// Mitsubishi GX Works2 project: PLC_GROUP2   PLC: FX3G

// global labels: Global1
VAR_GLOBAL
  SW10 AT X010 : BOOL;
END_VAR
VAR_GLOBAL CONSTANT
  chocolate : REAL := 1200;
  nuts : REAL := 300;
END_VAR
VAR_GLOBAL
  Dnuts AT D3100 : REAL;
END_VAR
VAR_GLOBAL CONSTANT
  pist : REAL := 300;
END_VAR
VAR_GLOBAL
  Dpist AT D3200 : REAL;
END_VAR
VAR_GLOBAL CONSTANT
  kad : REAL := 120;
END_VAR
VAR_GLOBAL
  SW1 AT X001 : BOOL;
  LAMP1 AT Y001 : BOOL;
END_VAR
VAR_GLOBAL CONSTANT
  melt_conts : REAL := 400;
END_VAR
VAR_GLOBAL
  Dchoco AT D3000 : REAL;
  Dkad AT D3300 : REAL;
END_VAR
VAR_GLOBAL CONSTANT
  meltTime : INT := 45;
END_VAR
VAR_GLOBAL
  meltingIndicator AT Y001 : BOOL;
  meltCoil AT TC1 : BOOL;
  SW07 AT X007 : BOOL;
  DAY_STARTED AT Y007 : BOOL;
  Dmelt AT D3400 : REAL;
  meltingprocess AT Y001 : BOOL;
  timeend AT M1 : BOOL;
  Dchocofill AT D2000 : REAL;
  Dnutsfill AT D2010 : REAL;
  Dpistfill AT D2020 : REAL;
  Dkadfill AT D2030 : REAL;
  StartDay AT Y007 : BOOL;
  shutDown AT X005 : BOOL;
  melting AT Y001 : BOOL;
  maxTemp AT X002 : BOOL;
  Lowchoco AT Y007 : BOOL;
  moldsCheck AT X003 : BOOL;
  moldCounter AT CC1 : BOOL;
END_VAR
VAR_GLOBAL CONSTANT
  CValue : INT := 4;
END_VAR
VAR_GLOBAL
  moldsIndicator AT CS1 : BOOL;
  castIndicator AT TS1 : BOOL;
END_VAR
VAR_GLOBAL CONSTANT
  castingTime : INT := 50;
END_VAR
VAR_GLOBAL
  casting AT Y002 : BOOL;
  movedToCasting AT M2 : BOOL;
  finishedCsting AT M3 : BOOL;
END_VAR
VAR_GLOBAL CONSTANT
  CastTime : WORD := 40;
END_VAR
VAR_GLOBAL
  cremeFilling AT X004 : BOOL;
  save_analog_1 AT D8201 : REAL;
END_VAR
VAR_GLOBAL CONSTANT
  input : REAL := 5;
END_VAR
VAR_GLOBAL
  isDubai AT M4 : BOOL;
  isNutsCream AT M4 : BOOL;
END_VAR
VAR_GLOBAL CONSTANT
  nutsForNutsChochlate : REAL := 100;
  pistForNutsChocholate : REAL := 100;
END_VAR
VAR_GLOBAL
  typeCheck AT M5 : BOOL;
END_VAR
VAR_GLOBAL CONSTANT
  pistForNutsChochlate : REAL := 100;
  nutsForDubai : REAL := 20;
  pistForDubai : REAL := 120;
  kadForDubai : REAL := 60;
END_VAR
VAR_GLOBAL
  finishedProdChoosing AT M6 : BOOL;
END_VAR
VAR_GLOBAL CONSTANT
  DivConst : REAL := 400;
END_VAR
VAR_GLOBAL
  LoopLamp AT M7 : BOOL;
  timeForY3 AT TC2 : BOOL;
END_VAR
VAR_GLOBAL CONSTANT
  Tvalue1 : INT := 5;
END_VAR
VAR_GLOBAL
  Y3Timer AT TS2 : BOOL;
  FillIndicator1 AT Y003 : BOOL;
  timeForY4 AT TC3 : BOOL;
END_VAR
VAR_GLOBAL CONSTANT
  Tvalue2 : INT := 5;
END_VAR
VAR_GLOBAL
  Y4Timer AT TS3 : BOOL;
  FillIndicator2 AT Y004 : BOOL;
  analog_input_1 : INT;
  analog_input AT D8280 : INT;
  FillIngTimer AT TC6 : BOOL;
END_VAR
VAR_GLOBAL CONSTANT
  FillingDuration : INT := 50;
END_VAR
VAR_GLOBAL
  fillingCreamIndicator AT TS6 : BOOL;
  StartFreezing AT X006 : BOOL;
  FreezingTimer AT TC7 : BOOL;
END_VAR
VAR_GLOBAL CONSTANT
  FreezingValue : INT := 30;
END_VAR
VAR_GLOBAL
  freezingLamp AT Y006 : BOOL;
  freezingIndicator AT TS7 : BOOL;
  finishedFillingInciator AT M8 : BOOL;
  finishedFrezingindicator AT M9 : BOOL;
  packingInit AT X000 : BOOL;
  packingLamp AT Y005 : BOOL;
  packingCount AT CC2 : BOOL;
  packingCounterIndicator AT CS2 : BOOL;
  finishedPacking AT M10 : BOOL;
  packageContainer AT D4000 : REAL;
END_VAR
VAR_GLOBAL CONSTANT
  packegeConst : REAL := 1;
END_VAR
VAR_GLOBAL
  cs2 AT CS2 : BOOL;
  finishedLoop AT M11 : BOOL;
END_VAR
VAR_GLOBAL CONSTANT
  chocoNeed : REAL := 400;
  nutsNeed : REAL := 100;
  pistNeed : REAL := 120;
  kadNeed : REAL := 60;
END_VAR
VAR_GLOBAL
  outOfStock AT M12 : BOOL;
  DayEnded AT M13 : BOOL;
END_VAR
VAR_GLOBAL CONSTANT
  multiplyConstant : REAL := 40;
END_VAR
VAR_GLOBAL
  analog_output AT D8282 : INT;
  emptyReg AT D7000 : REAL;
END_VAR
VAR_GLOBAL CONSTANT
  zeroConst : REAL;
  zeroValue : INT;
END_VAR
VAR_GLOBAL
  inventoryCheck AT M15 : BOOL;
  movedStock AT M17 : BOOL;
END_VAR

// task Task_01 (event TRUE, interval 0, priority 31): POU_01

PROGRAM POU_01
VAR CONSTANT
  choco : REAL := 400;
END_VAR
(* structured ladder/FBD written out as ST: instructions are called as NAME(EN, inputs, outputs); _pN, _eN, _tN stand for wires *)
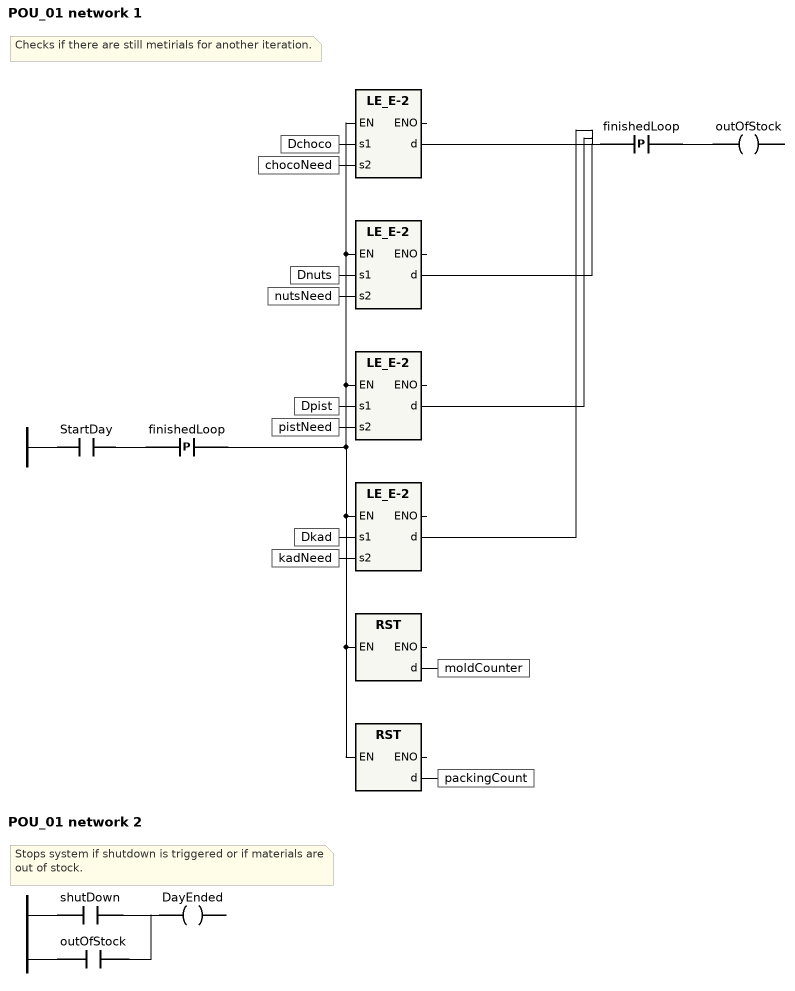
(* network 1 *)
(* Checks if there are still metirials for another iteration. *)
_p1 := StartDay AND LDP(TRUE, finishedLoop);
LE_E(_p1, Dchoco, chocoNeed, _t2);
LE_E(_p1, Dnuts, nutsNeed, _t3);
LE_E(_p1, Dpist, pistNeed, _t4);
LE_E(_p1, Dkad, kadNeed, _t5);
outOfStock := (_t2 OR _t3 OR _t4 OR _t5) AND LDP(TRUE, finishedLoop);
RST(_p1, moldCounter);
RST(_p1, packingCount);
(* network 2 *)
(* Stops system if shutdown is triggered or if materials are out of stock. *)
DayEnded := shutDown OR outOfStock;
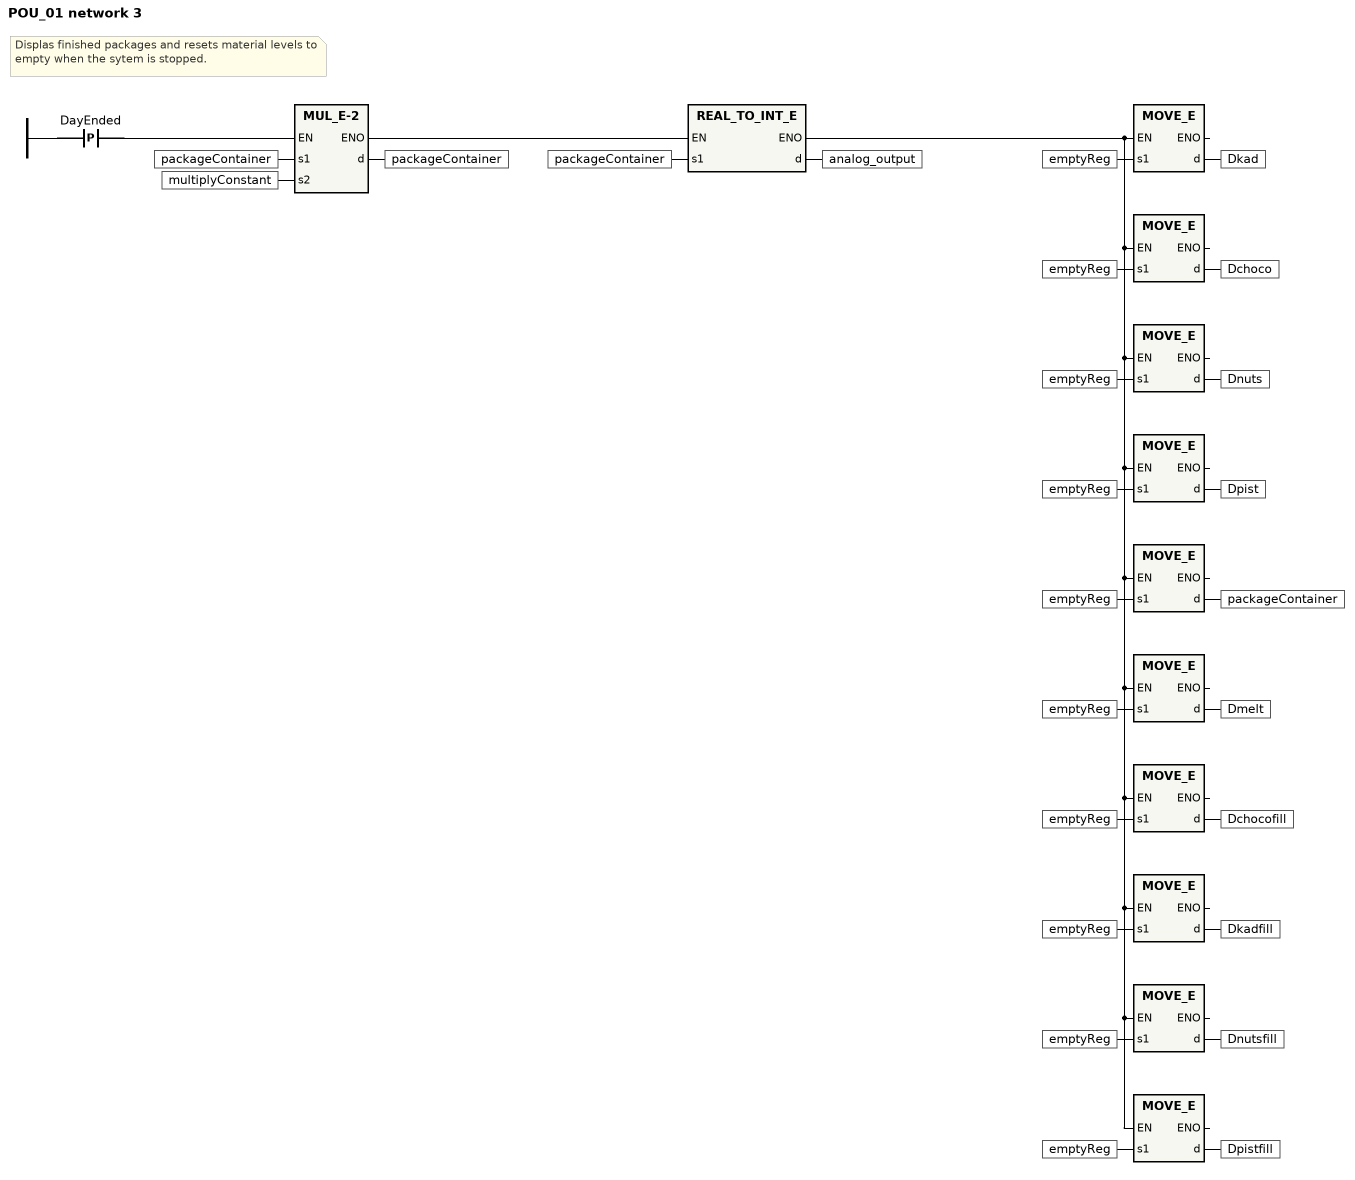
(* network 3 *)
(* Displas finished packages and resets material levels to empty when the sytem is stopped. *)
_e1 := MUL_E(LDP(TRUE, DayEnded), packageContainer, multiplyConstant, packageContainer);
_e2 := REAL_TO_INT_E(_e1, packageContainer, analog_output);
MOVE_E(_e2, emptyReg, Dkad);
MOVE_E(_e2, emptyReg, Dchoco);
MOVE_E(_e2, emptyReg, Dnuts);
MOVE_E(_e2, emptyReg, Dpist);
MOVE_E(_e2, emptyReg, packageContainer);
MOVE_E(_e2, emptyReg, Dmelt);
MOVE_E(_e2, emptyReg, Dchocofill);
MOVE_E(_e2, emptyReg, Dkadfill);
MOVE_E(_e2, emptyReg, Dnutsfill);
MOVE_E(_e2, emptyReg, Dpistfill);
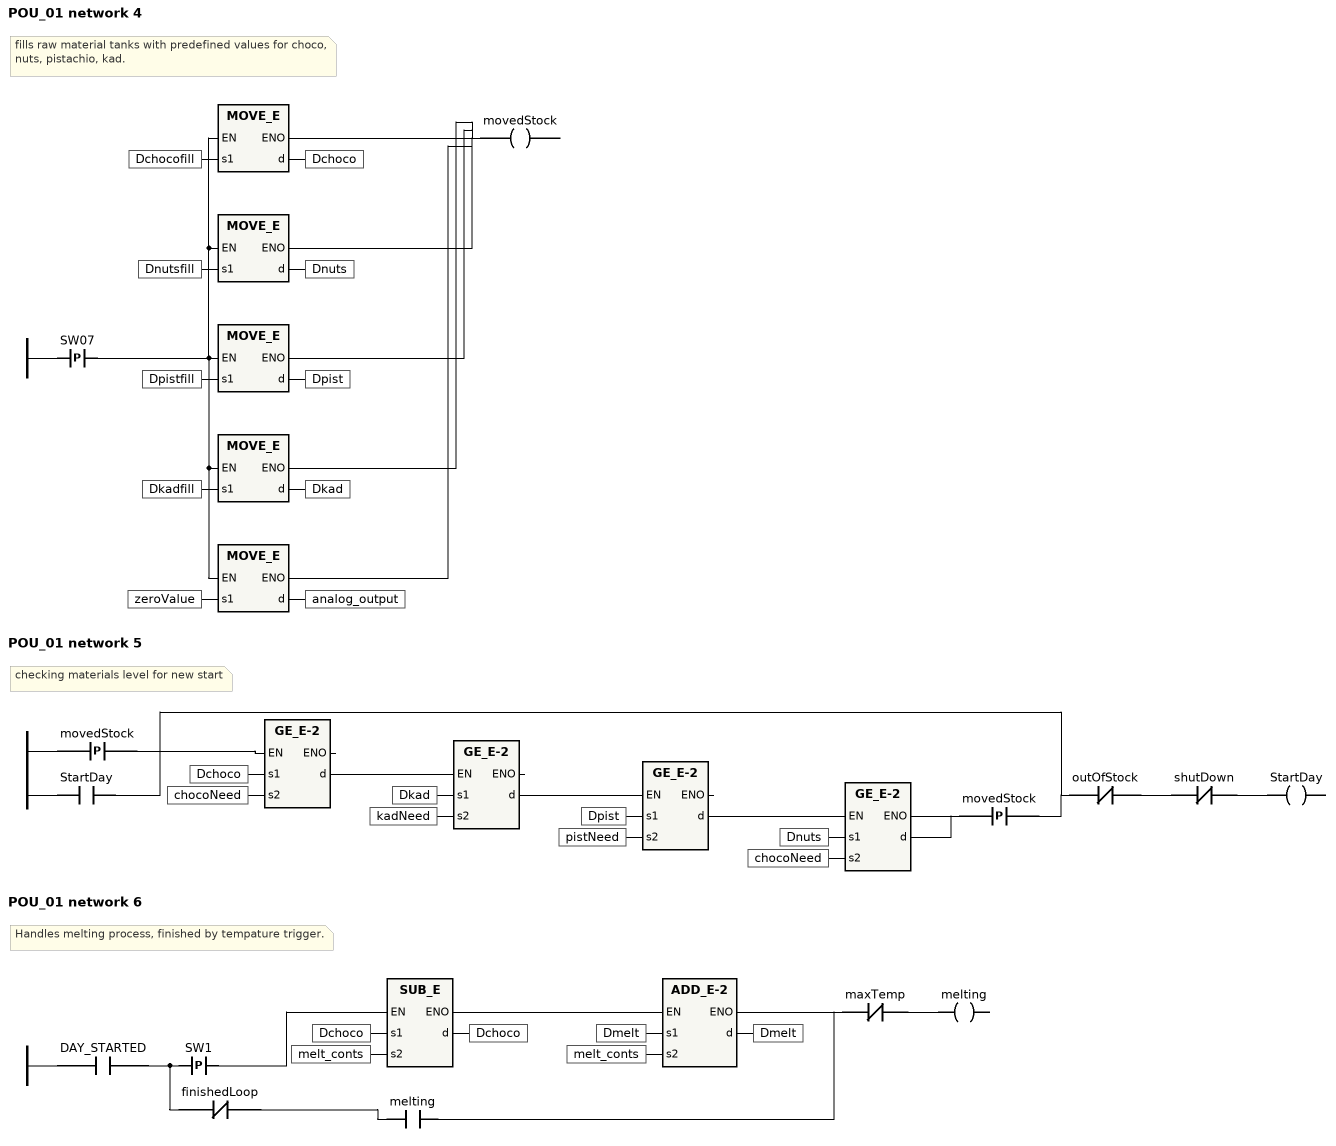
(* network 4 *)
(* fills raw material tanks with predefined values for choco, nuts, pistachio, kad. *)
_p1 := LDP(TRUE, SW07);
_e2 := MOVE_E(_p1, Dchocofill, Dchoco);
_e3 := MOVE_E(_p1, Dnutsfill, Dnuts);
_e4 := MOVE_E(_p1, Dpistfill, Dpist);
_e5 := MOVE_E(_p1, Dkadfill, Dkad);
_e6 := MOVE_E(_p1, zeroValue, analog_output);
movedStock := _e2 OR _e3 OR _e4 OR _e5 OR _e6;
(* network 5 *)
(* checking materials level for new start *)
GE_E(LDP(TRUE, movedStock), Dchoco, chocoNeed, _t1);
GE_E(_t1, Dkad, kadNeed, _t2);
GE_E(_t2, Dpist, pistNeed, _t3);
_e5 := GE_E(_t3, Dnuts, chocoNeed, _t4);
StartDay := ((((_e5 OR _t4) AND LDP(TRUE, movedStock)) OR StartDay) AND NOT outOfStock) AND NOT shutDown;
(* network 6 *)
(* Handles melting process, finished by tempature trigger. *)
_e1 := SUB_E(DAY_STARTED AND LDP(TRUE, SW1), Dchoco, melt_conts, Dchoco);
_e2 := ADD_E(_e1, Dmelt, melt_conts, Dmelt);
melting := (_e2 OR (DAY_STARTED AND NOT finishedLoop AND melting)) AND NOT maxTemp;
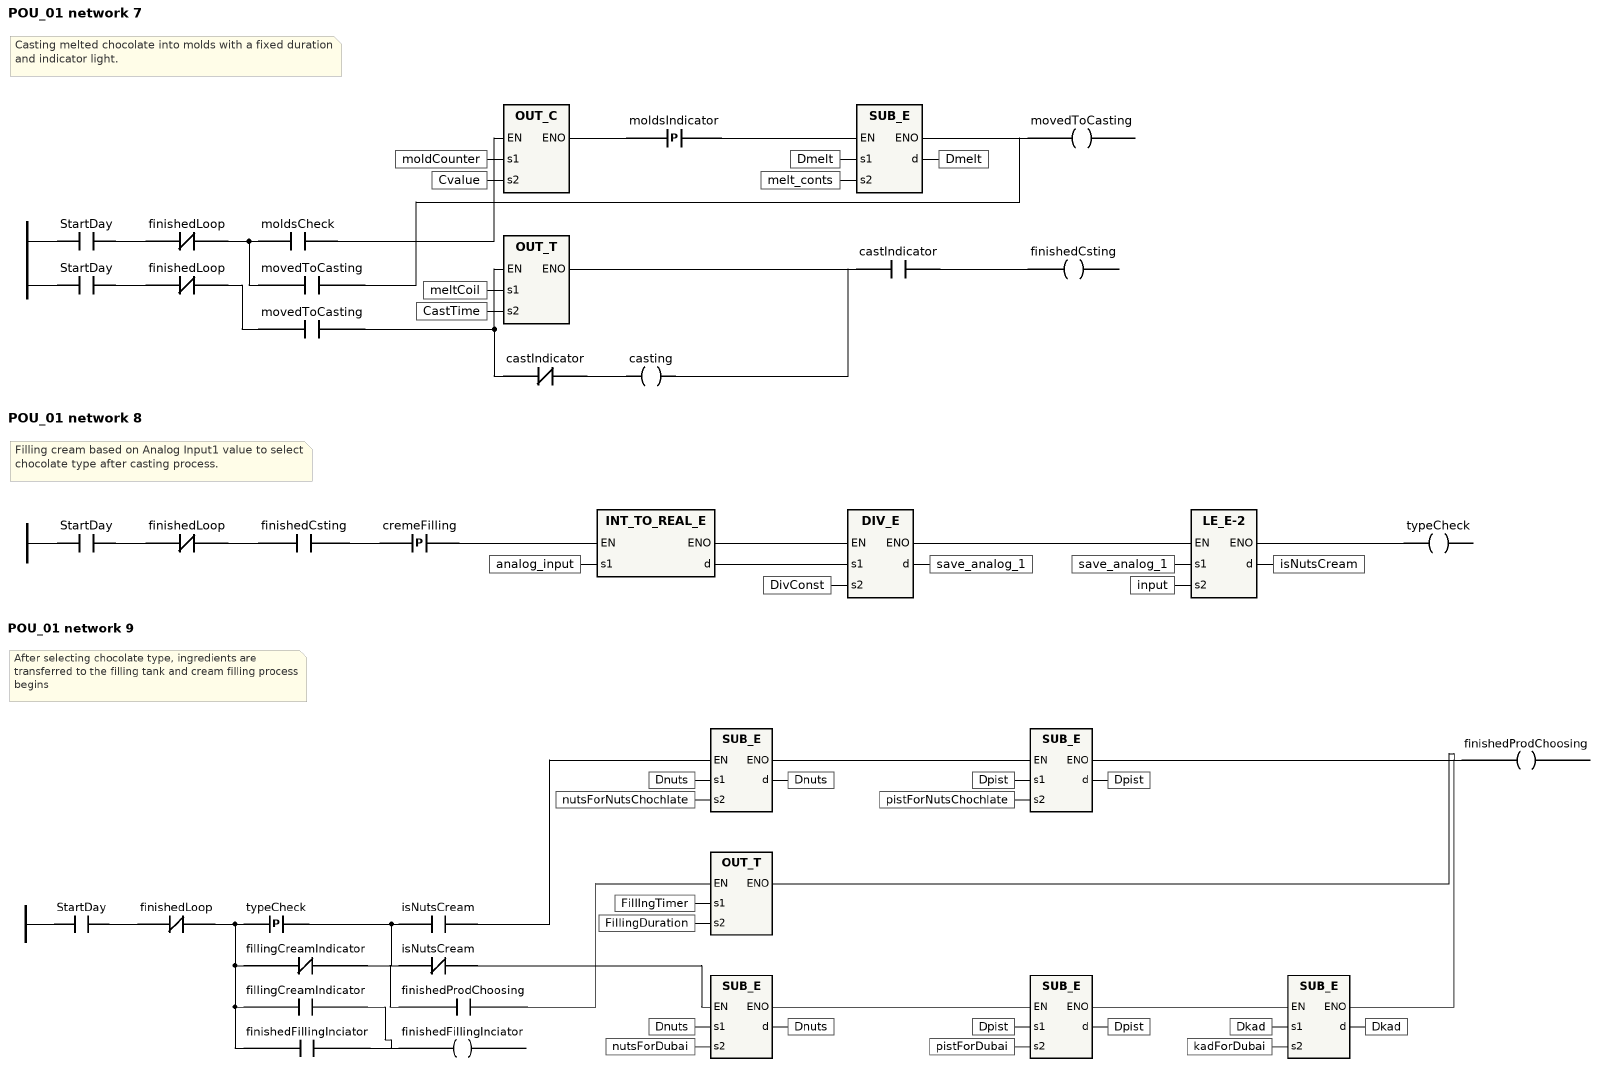
(* network 7 *)
(* Casting melted chocolate into molds with a fixed duration and indicator light. *)
_p1 := StartDay AND NOT finishedLoop;
_e2 := OUT_C(_p1 AND moldsCheck, moldCounter, Cvalue);
_e3 := SUB_E(_e2 AND LDP(TRUE, moldsIndicator), Dmelt, melt_conts, Dmelt);
movedToCasting := _e3 OR (_p1 AND movedToCasting);
_p4 := StartDay AND NOT finishedLoop AND movedToCasting;
_e5 := OUT_T(_p4, meltCoil, CastTime);
_p6 := _p4 AND NOT castIndicator;
casting := _p6;
finishedCsting := (_e5 OR _p6) AND castIndicator;
(* network 8 *)
(* Filling cream based on Analog Input1 value to select chocolate type after casting process. *)
_e2 := INT_TO_REAL_E(StartDay AND NOT finishedLoop AND finishedCsting AND LDP(TRUE, cremeFilling), analog_input, _t1);
_e3 := DIV_E(_e2, _t1, DivConst, save_analog_1);
_e4 := LE_E(_e3, save_analog_1, input, isNutsCream);
typeCheck := _e4;
(* network 9 *)
(* After selecting chocolate type, ingredients are transferred to the filling tank and cream filling process begins *)
_p1 := StartDay AND NOT finishedLoop;
_p2 := _p1 AND LDP(TRUE, typeCheck);
_e3 := SUB_E(_p2 AND isNutsCream, Dnuts, nutsForNutsChochlate, Dnuts);
_e4 := SUB_E(_e3, Dpist, pistForNutsChochlate, Dpist);
_e5 := SUB_E(_p2 AND NOT isNutsCream, Dnuts, nutsForDubai, Dnuts);
_e6 := SUB_E(_e5, Dpist, pistForDubai, Dpist);
_e7 := SUB_E(_e6, Dkad, kadForDubai, Dkad);
_e8 := OUT_T(_p1 AND NOT fillingCreamIndicator AND finishedProdChoosing, FillIngTimer, FillingDuration);
finishedProdChoosing := _e4 OR _e7 OR _e8;
finishedFillingInciator := (_p1 AND fillingCreamIndicator) OR (_p1 AND finishedFillingInciator);
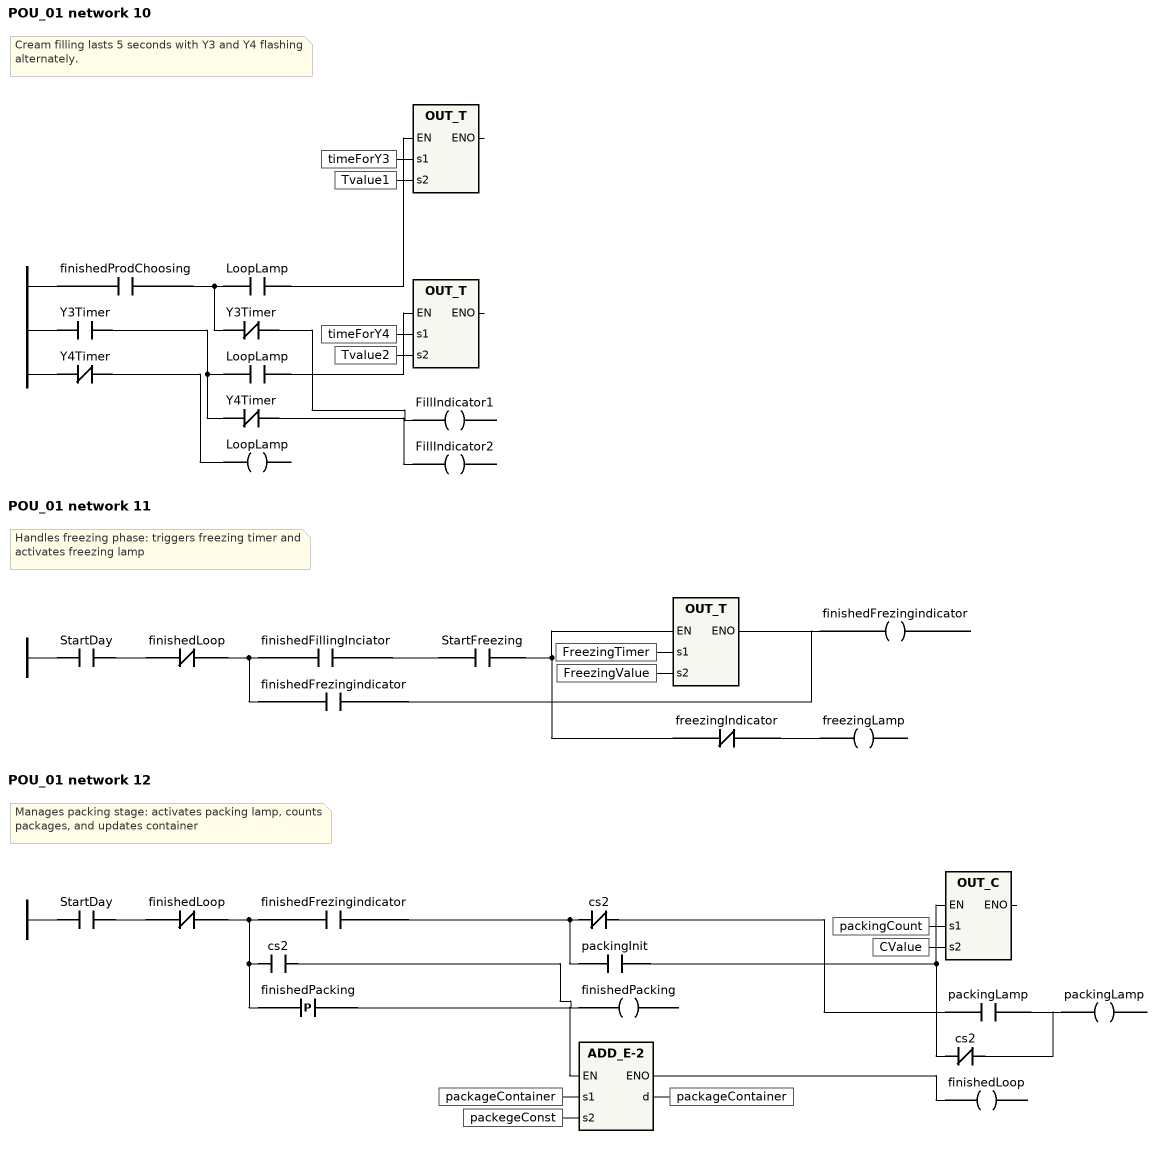
(* network 10 *)
(* Cream filling lasts 5 seconds with Y3 and Y4 flashing alternately. *)
OUT_T(finishedProdChoosing AND LoopLamp, timeForY3, Tvalue1);
FillIndicator1 := finishedProdChoosing AND NOT Y3Timer;
OUT_T(Y3Timer AND LoopLamp, timeForY4, Tvalue2);
FillIndicator2 := Y3Timer AND NOT Y4Timer;
LoopLamp := NOT Y4Timer;
(* network 11 *)
(* Handles freezing phase: triggers freezing timer and activates freezing lamp *)
_p1 := StartDay AND NOT finishedLoop;
_p2 := _p1 AND finishedFillingInciator AND StartFreezing;
_e3 := OUT_T(_p2, FreezingTimer, FreezingValue);
finishedFrezingindicator := _e3 OR (_p1 AND finishedFrezingindicator);
freezingLamp := _p2 AND NOT freezingIndicator;
(* network 12 *)
(* Manages packing stage: activates packing lamp, counts packages, and updates container *)
_p1 := StartDay AND NOT finishedLoop;
_p2 := _p1 AND finishedFrezingindicator;
_p3 := _p2 AND packingInit;
packingLamp := (_p2 AND NOT cs2 AND packingLamp) OR (_p3 AND NOT cs2);
OUT_C(_p3, packingCount, CValue);
finishedPacking := _p1 AND cs2;
_e4 := ADD_E(_p1 AND LDP(TRUE, finishedPacking), packageContainer, packegeConst, packageContainer);
finishedLoop := _e4;
END_PROGRAM
